// TwinCAT 3 PLC project EncoderLogger
// ProgramVersion: 3.1.4022.2
// libraries:
//   Tc2_EtherCAT, * (Beckhoff Automation GmbH)
//   Tc2_Standard, * (Beckhoff Automation GmbH)
//   Tc2_System, * (Beckhoff Automation GmbH)
//   Tc2_Utilities, * (Beckhoff Automation GmbH)
//   Tc3_Module, * (Beckhoff Automation GmbH)
//   VisuSymbols,3.5.10.0,System
// project tree:
//   DUTs/ DCTIME64_UINT.TcDUT
//   / GlobalTextList.TcGTLO, PlcTask.TcTTO (not stored), Visualization Manager.TcVMO (not stored)
//   POUs/ GENERATE_FILENAME.TcPOU, MAIN.TcPOU
//   VISUs/ Visualization.TcVIS
// real-time tasks:
//   TASK PlcTask: cycle T#100us, priority 20, ADS port 350
// I/O:
//   DEVICE Device 1 (EtherCAT), AmsNetId 5.49.22.42.2.1
//     Term 1 (EK1200) [EK1200-5000 EtherCAT Power supply (2A E-Bus)]
//       Term 2 (EL5101) [EL5101 1Ch. Inc. Encoder 5V]
//       Term 3 (EL9011) [EL9011 End Terminal]
// variable links:
//   EncoderLogger Instance <-> Device 1 (EtherCAT)/Term 1 (EK1200)/Term 2 (EL5101)
//     PlcTask Inputs/MAIN.enc_raw <-> ENC Status compact/Counter value

// ---- DUTs/DCTIME64_UINT.TcDUT
TYPE DCTIME64_UINT :
STRUCT
	tDC : T_DCTIME64;
	iData : UINT;
END_STRUCT
END_TYPE

// ---- POUs/GENERATE_FILENAME.TcPOU
FUNCTION GENERATE_FILENAME : STRING
VAR_INPUT
	sPrefix : STRING;
	stTime : TIMESTRUCT;
	sSuffix : STRING;
END_VAR
VAR
	sOutput : STRING;
	sTime : STRING;
END_VAR

sTime := SYSTEMTIME_TO_STRING(stTime);

sOutput := sPrefix;

//sOutput := CONCAT(sOutput, 'test');

sOutput := CONCAT(sOutput, LEFT(sTime, 10));

sOutput := CONCAT(sOutput, ' ');
sOutput := CONCAT(sOutput, MID(sTime, 2, 12));
sOutput := CONCAT(sOutput, '-');
sOutput := CONCAT(sOutput, MID(sTime, 2, 15));
sOutput := CONCAT(sOutput, '-');
sOutput := CONCAT(sOutput, MID(sTime, 2, 18));

sOutput := CONCAT(sOutput, sSuffix);

GENERATE_FILENAME := sOutput;

END_FUNCTION

// ---- POUs/MAIN.TcPOU
PROGRAM MAIN
VAR
	heartbeat 		: UDINT;
	
	enc_raw AT %I* 	: UINT;
	enc_angle 		: REAL;
	
	// Time
	tDC 			: T_DCTIME64;
	sTime 			: STRING;
	dDate 			: TIMESTRUCT;
	
	// File writing
	bRecordData 	: BOOL;
	iFileState 		: UINT;
	sFilePath 		: STRING 	:= 'C:\Users\Public\Documents\EncoderData\';
	sFileType		: STRING	:= '.bin';
	sFileName		: STRING;
	fbRecordTrigger	: R_TRIG;
	
	fbFileOpen		: FB_FileOpen; 				// Opens file
	fbFileClose		: FB_FileClose;				// Closes file
	fbFileWriter	: FB_FileWrite;				// Writes binary
	
	bBusy			: BOOL;
	bError			: BOOL;
	nErrId			: UDINT;
	hFile			: UINT		:= 0;
	
	// Buffer
	stBuffer 		: ARRAY [0..iBufferLength] OF DCTIME64_UINT;	// Buffer to dump data into
	iEndOfBuffer	: UDINT		:= 0;								// Index of the end of the buffer
	bBufferFull 	: BOOL;											// Is stBuffer full?
	stBufferToWrite	: ARRAY [0..iBufferLength] OF DCTIME64_UINT;	// Buffer to write into file (static copy of stBuffer)
	iLenToWrite     : UDINT;										// Number of elements in stBufferToWrite

END_VAR
VAR CONSTANT
	iBufferLength	: UDINT		:= 50;								// Number of elements in the array
	cbElementSize 	: UDINT		:= SIZEOF(DCTIME64_UINT);			// Size of each element
END_VAR

heartbeat := heartbeat + 1;

// Get the encoder value
enc_angle := enc_raw MOD (360*4);
enc_angle := enc_angle / 4;


// Get the time
tDC := F_GetCurDcTaskTime64();
sTime := DCTIME64_TO_STRING(tDC);
dDate := DCTIME64_TO_SYSTEMTIME(tDC);


// Clear the buffer and set the file name when we start recording
fbRecordTrigger(CLK:=bRecordData);
IF fbRecordTrigger.Q THEN
	MEMSET( destAddr := ADR(stBuffer),
			fillByte := 0,
			n := cbElementSize * iBufferLength);
	iEndOfBuffer := 0;
	
	sFileName := GENERATE_FILENAME(sFilePath, dDate, sFileType);
END_IF


// If we're recording, and there's still room, add a new element to the buffer
IF bRecordData AND NOT bBufferFull THEN
	stBuffer[iEndOfBuffer].tDC := tDC;
	stBuffer[iEndOfBuffer].iData := enc_raw;
	
	iEndOfBuffer := iEndOfBuffer + 1;	
END_IF


// Check if the buffer is full
IF iBufferLength > iEndOfBuffer THEN
	bBufferFull := FALSE;
ELSE
	bBufferFull := TRUE;
END_IF


// State machine to handle writing the file
CASE iFileState OF
	0:	// Wait to start
		IF bRecordData THEN
			bBusy := TRUE;
			
			// Reset variables
			bError	:= FALSE;
			nErrId	:= 0;
			hFile	:= 0;
			
			iFileState := 10;
		END_IF
		
	10:	// Open the file
		fbFileOpen(bExecute := FALSE);
		fbFileOpen(	sNetId := '', 
					sPathName := sFileName, 
					nMode := FOPEN_MODEWRITE OR FOPEN_MODEBINARY, 
					ePath := PATH_GENERIC, 
					bExecute := TRUE);
		iFileState := 20;
	
	20:	// Wait for opening to finish
		fbFileOpen(bExecute := FALSE, bError => bError, nErrID => nErrID, hFile => hFile );
		IF NOT fbFileOpen.bBusy THEN
			IF NOT fbFileOpen.bError THEN
				iFileState := 30;
			ELSE
				// Error: file not found?
				iFileState := 100;
			END_IF
		END_IF
		
	30: // If we still want to write the file, write it
		IF bRecordData THEN
			// Clear stBufferToWrite				
			MEMSET( destAddr := ADR(stBufferToWrite),
					fillByte := 0,
					n := cbElementSize * iBufferLength);
		    
			// Copy the stBuffer into stBufferToWrite
			MEMCPY(	srcAddr := ADR(stBuffer),
					destAddr := ADR(stBufferToWrite),
					n := iEndOfBuffer * cbElementSize);
			
			// Write stBufferToWrite into the file
			fbFileWriter( sNetId := '',
						hFile := hFile,
						pWriteBuff := ADR(stBufferToWrite),
						cbWriteLen := iEndOfBuffer * cbElementSize,
						bExecute := TRUE);
			
			// Store the number of elements being written
			iLenToWrite := iEndOfBuffer;
			
			// Clear stBuffer						
			MEMSET( destAddr := ADR(stBuffer),
					fillByte := 0,
					n := cbElementSize * iBufferLength);
			iEndOfBuffer := 0;
			
			iFileState := 40;
		
		ELSE // Stop writing
			iFileState := 200;
		END_IF
		
	40:	// Wait for the write to finish
		fbFileWriter( bExecute := FALSE, bError => bError, nErrID => nErrID );
		IF NOT fbFileWriter.bBusy THEN
			IF NOT fbFileWriter.bError THEN
				iFileState := 30;(* Write next record *)
			ELSE(* Error *)
				iFileState := 100;
			END_IF
		END_IF
			
	100: // Error
		IF ( hFile <> 0 ) THEN
			iFileState := 200; (* Close the source file *)
		ELSE
			bBusy := FALSE;
			iFileState := 0;	(* Ready *)
		END_IF
		
	200: // Close
		fbFileClose( bExecute := FALSE );
		fbFileClose( sNetId := '', hFile := hFile, bExecute := TRUE );
		iFileState := 210;
		
	210: // Wait for close to finish
		fbFileClose( bExecute := FALSE, bError => bError, nErrID => nErrID );
		IF ( NOT fbFileClose.bBusy ) THEN
			hFile := 0;
			bBusy := FALSE;
			iFileState := 0;	(* Ready *)
		END_IF

END_CASE

END_PROGRAM

// ---- GlobalTextList.TcGTLO
TEXTLIST GlobalTextList
  592 = 'File: %s'
  936 = 'iFileState: %d'
  594 = 'Raw: %s'
  320 = 'Raw: %s\n\n'
  207 = 'Raw: %s\n\n\n\n'
  685 = 'Recording? %s'
  102 = 'Time: %s'
  113 = 'Write'
END_TEXTLIST

// ---- VISUs/Visualization.TcVIS
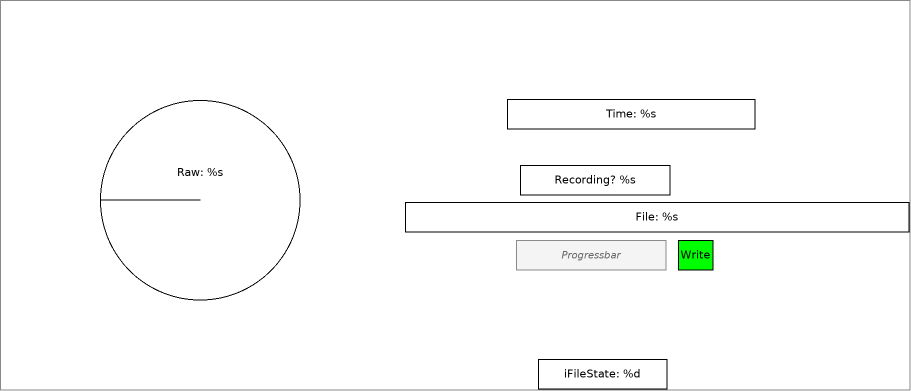
VISUALIZATION Visualization  // 911x391
    Rectangle (520,165 150x30), "Recording? %s", text variable: MAIN.bRecordData
        OnMouseDown: execute { MAIN.bRecordData := NOT MAIN.bRecordData; }
    Ellipse (100,100 200x200), "Raw: %s", text variable: MAIN.enc_raw
    Line (200,200) (100,200)
        p2858320360: MAIN.enc_angle
    Progressbar (516,240 150x30), variable: MAIN.iEndOfBuffer
    Rectangle (678,240 35x30), "Write", text variable: MAIN.bRecordData, invisible if: not MAIN.fbFileWriter.bBusy
    Rectangle (538,359 129x30), "iFileState: %d", text variable: MAIN.iFileState
    Rectangle (507,99 248x30), "Time: %s", text variable: MAIN.sTime
    Rectangle (405,202 504x30), "File: %s", text variable: MAIN.sFileName
END_VISUALIZATION
